FUNCTION IncULINT : ULINT		// Increments the given ULINT value
VAR_IN_OUT
	ioNum:	ULINT;		// Value to increment
END_VAR

IncULINT := ioNum := ioNum + 1;

END_FUNCTION

(* stored: Version 1.1.0.1, ProductVersion 3.1.4026.18
   POU IncULINT: Id {2e5640c3-7558-4a4c-9b21-818e0f3756e0}, SpecialFunc None *)
